# EPICS autosave request: iocBoot/gmca_23o_ioc1/dbSave/auto_settings.req
%
file BP_Hd1_.req P=23o:
file BP_Hd2_.req P=23o:
file BP_Hd3_.req P=23o:
file BP_Kb_.req  P=23o:
file BP_Mo_.req  P=23o:
file CS_Ah_.req  P=23o:
file CS_Av_.req  P=23o:
file HD_Dn_.req  P=23o:
file HD_Up_.req  P=23o:
file HD_St_.req  P=23o:
file KB_Hy_.req  P=23o:
file KB_Hz_.req  P=23o:
file KB_Vy_.req  P=23o:
file KB_Vz_.req  P=23o:
file MO_En_.req  P=23o:
file MO_Ps_.req  P=23o:
file MO_Tn1_.req P=23o:
file MO_Tn2_.req P=23o:
file WS_Ah_.req  P=23o:
file WS_Av_.req  P=23o:
%
% file keithleys.req P=23o:
%

file DAC128_single.req P=23o:,D=1,N=1
file DAC128_single.req P=23o:,D=1,N=2
file DAC128_single.req P=23o:,D=1,N=3
file DAC128_single.req P=23o:,D=1,N=4
file DAC128_single.req P=23o:,D=1,N=5
file DAC128_single.req P=23o:,D=1,N=6
file DAC128_single.req P=23o:,D=1,N=7
file DAC128_single.req P=23o:,D=1,N=8

file DAC128_single.req P=23o:,D=2,N=1
file DAC128_single.req P=23o:,D=2,N=2
file DAC128_single.req P=23o:,D=2,N=3
file DAC128_single.req P=23o:,D=2,N=4
file DAC128_single.req P=23o:,D=2,N=5
file DAC128_single.req P=23o:,D=2,N=6
file DAC128_single.req P=23o:,D=2,N=7
file DAC128_single.req P=23o:,D=2,N=8
file DAC128_single.req P=23o:,D=2,N=9
file DAC128_single.req P=23o:,D=2,N=10
file DAC128_single.req P=23o:,D=2,N=11
file DAC128_single.req P=23o:,D=2,N=12
file DAC128_single.req P=23o:,D=2,N=13
file DAC128_single.req P=23o:,D=2,N=14
file DAC128_single.req P=23o:,D=2,N=15
file DAC128_single.req P=23o:,D=2,N=16

% file digital_IO_16_desc.req P=23o:bo0:ch
% file digital_IO_24_desc.req P=23o:pmac20:acc65e:bo
% file digital_IO_24_desc.req P=23o:pmac21:acc65e:bo
